{attribute addProperty BoxType "EJ3004-0000-0019"}
{attribute addProperty Id "StatusAT %I*Status_C6F82E6F1621ValueAT %I*INT16217"}
{attribute addProperty CRC "1466166969"}
{attribute addProperty SizeInBites "32"}
{attribute addProperty SizeInBytes "4"}
TYPE AI_Standard_Channel_5763EEB9 :
STRUCT
	{attribute addProperty Name "Status"}
	Status AT %I* : Status_C6F82E6F;
	{attribute addProperty Name "Value"}
	Value AT %I* : INT;
END_STRUCT
END_TYPE

(* stored: Version 1.2.0.0, ProductVersion 3.1.4024.9
   DUT AI_Standard_Channel_5763EEB9: Id {8c950b2c-4d18-4a44-abf0-dc7744f2cf51} *)
